Omron CX-Programmer project NewProject (CX-Programmer 9.61)

# PLC TrialGITHUB: CJ1M CPU11

## Program NewProgram1 (cyclic task 0)

### Section Section1

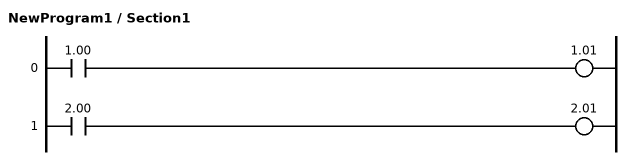
; rung 0
LD 1.00
OUT 1.01
; rung 1
LD 2.00
OUT 2.01

### Section END
; rung 0
END(001)